FUNCTION_BLOCK inicializarPosOcupEstanteria
VAR_INPUT
END_VAR
VAR_OUTPUT
END_VAR
VAR
	i: INT;
	fila: INT;
	col: INT;
END_VAR

// Se inicializan las posicones del amlmcen a false
// por defecto se empieza con el almacen vacio
FOR fila := 1 TO 6 DO
    FOR col := 1 TO 3 DO
        // la primera posicion libre 
		 GVLvar.baldasOcupadas[fila,col] := FALSE;
    END_FOR
END_FOR

END_FUNCTION_BLOCK

(* stored: Version 1.1.0.1, ProductVersion 3.1.4024.15
   POU inicializarPosOcupEstanteria: Id {b4946830-5ebd-495b-81cc-70df109f41ee}, SpecialFunc None *)
